{attribute 'qualified_only'}
{attribute 'strict'}
{attribute 'to_string'}
TYPE E_Status :
(
	//Actual Pulse Power State
	SAFE			:= 0, //IDLE
	CHARGING		:= 1, //Charge
	CHARGECOMPLETE	:= 2, //EOC
	DISCONNECTING	:= 3, //Disconnect
	DUMPING			:= 4, 
	ABORT			:= 5,	
	TRIPPED			:= 6,
	LOCAL_MODE		:= 7
) ;
END_TYPE

(* stored: Version 1.1.0.1, ProductVersion 3.1.4024.11
   DUT E_Status: Id {ccb993a3-5d36-42c6-942b-dcc84eec1dde} *)
